// TIA Portal V18 export
// export: Created 2026-06-12T00:00:00Z, ExportSetting WithDefaults
DATA_BLOCK "Timer_Sim_DB"   // DB10
TITLE = Timer_Sim_DB
// DB chứa biến đếm thời gian cho khối mô phỏng
// stored: AutoNumber true, InstanceOfName IEC_TIMER, OfSystemLibElement IEC_TIMER, OfSystemLibVersion 1.0
"IEC_TIMER"
   // VAR
   //    PT : Time;
   //    ET { ExternalWritable := 'False'} : Time;
   //    IN : Bool;
   //    Q { ExternalWritable := 'False'} : Bool;
   // END_VAR
BEGIN
END_DATA_BLOCK
